// TIA Portal V17 export
// export: Created 2024-08-29T18:23:43.9089701Z, ExportSetting WithDefaults, DisplayName Totally Integrated Automation Portal, DisplayVersion V17 Update 7, DisplayName TIA Portal Openness, DisplayVersion V17 Update 7, DisplayName TIA Portal Version Control Interface, DisplayVersion V17, DisplayName SINAMICS Startdrive Advanced, DisplayVersion V17 SP2, DisplayName SINAMICS Startdrive G110M, G120, G120C, G120D, G120P, G115D, DisplayVersion V17 SP2, DisplayName SINAMICS Startdrive G130, G150, S120, S150, SINAMICS MV, S210, DisplayVersion V17 SP2, DisplayName STEP 7 Professional, DisplayVersion V17 Update 7, DisplayName STEP 7 Safety, DisplayVersion V17 Update 6, DisplayName WinCC Advanced / Unified PC, DisplayVersion V17 Update 7
FUNCTION "dcMotorControl" : Void   // FC20, LAD
{ S7_Optimized_Access := 'TRUE' }
VERSION : 0.1
// stored: AutoNumber true, IsIECCheckEnabled false, SetENOAutomatically false, UDAEnableTagReadback false
   VAR_TEMP   // added for the SCL form of the ladder/FBD networks
      _w1 : Bool;
      _w2 : Bool;
   END_VAR
BEGIN

REGION Network 1: SELECT MOTOR PARAMETERS
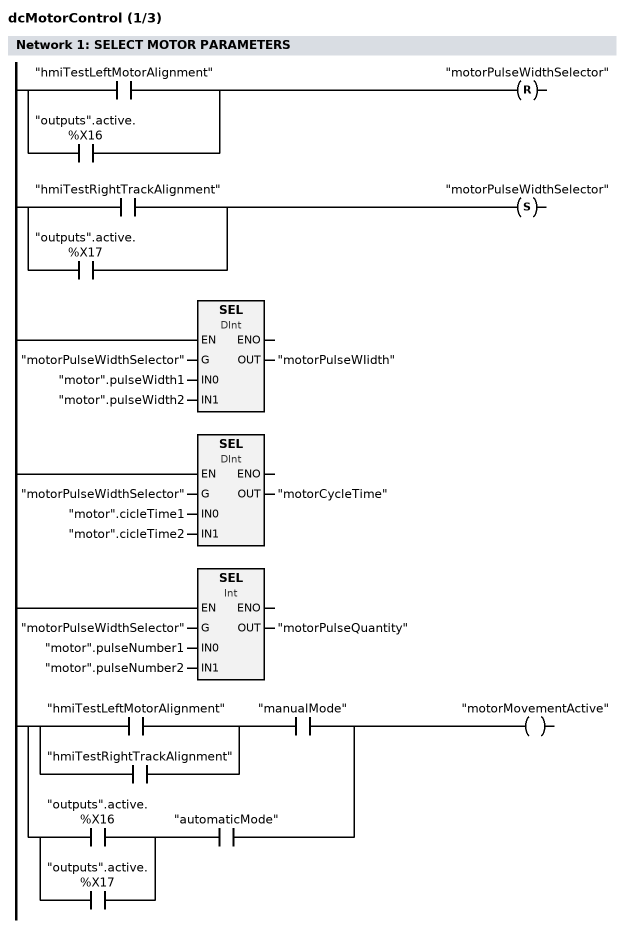
   RUNG wire#powerrail
      Contact( "hmiTestLeftMotorAlignment" )
      wire#w1
      R_Coil( "motorPulseWidthSelector" )
   END_RUNG
   RUNG wire#powerrail
      Contact( "outputs".active.%X16 )
   END_RUNG wire#w1
   RUNG wire#powerrail
      Contact( "hmiTestRightTrackAlignment" )
      wire#w2
      S_Coil( "motorPulseWidthSelector" )
   END_RUNG
   RUNG wire#powerrail
      Contact( "outputs".active.%X17 )
   END_RUNG wire#w2
   RUNG wire#powerrail
      { S7_Templates := "value_type := DInt" } SEL(g := "motorPulseWidthSelector", in0 := "motor".pulseWidth1, in1 := "motor".pulseWidth2, out => "motorPulseWIidth")
   END_RUNG
   RUNG wire#powerrail
      { S7_Templates := "value_type := DInt" } SEL(g := "motorPulseWidthSelector", in0 := "motor".cicleTime1, in1 := "motor".cicleTime2, out => "motorCycleTime")
   END_RUNG
   RUNG wire#powerrail
      { S7_Templates := "value_type := Int" } SEL(g := "motorPulseWidthSelector", in0 := "motor".pulseNumber1, in1 := "motor".pulseNumber2, out => "motorPulseQuantity")
   END_RUNG
   RUNG wire#powerrail
      Contact( "hmiTestLeftMotorAlignment" )
      wire#w3
      Contact( "manualMode" )
      wire#w4
      Coil( "motorMovementActive" )
   END_RUNG
   RUNG wire#powerrail
      Contact( "hmiTestRightTrackAlignment" )
   END_RUNG wire#w3
   RUNG wire#powerrail
      Contact( "outputs".active.%X16 )
      wire#w5
      Contact( "automaticMode" )
   END_RUNG wire#w4
   RUNG wire#powerrail
      Contact( "outputs".active.%X17 )
   END_RUNG wire#w5
   // the same network as SCL:
   IF "hmiTestLeftMotorAlignment" OR "outputs".active.%X16 THEN "motorPulseWidthSelector" := FALSE; END_IF;
   IF "hmiTestRightTrackAlignment" OR "outputs".active.%X17 THEN "motorPulseWidthSelector" := TRUE; END_IF;
   "motorPulseWIidth" := SEL(G := "motorPulseWidthSelector", IN0 := "motor".pulseWidth1, IN1 := "motor".pulseWidth2);
   "motorCycleTime" := SEL(G := "motorPulseWidthSelector", IN0 := "motor".cicleTime1, IN1 := "motor".cicleTime2);
   "motorPulseQuantity" := SEL(G := "motorPulseWidthSelector", IN0 := "motor".pulseNumber1, IN1 := "motor".pulseNumber2);
   "motorMovementActive" := (("hmiTestLeftMotorAlignment" OR "hmiTestRightTrackAlignment") AND "manualMode") OR (("outputs".active.%X16 OR "outputs".active.%X17) AND "automaticMode");
END_REGION

REGION Network 2: PWM CONTROL
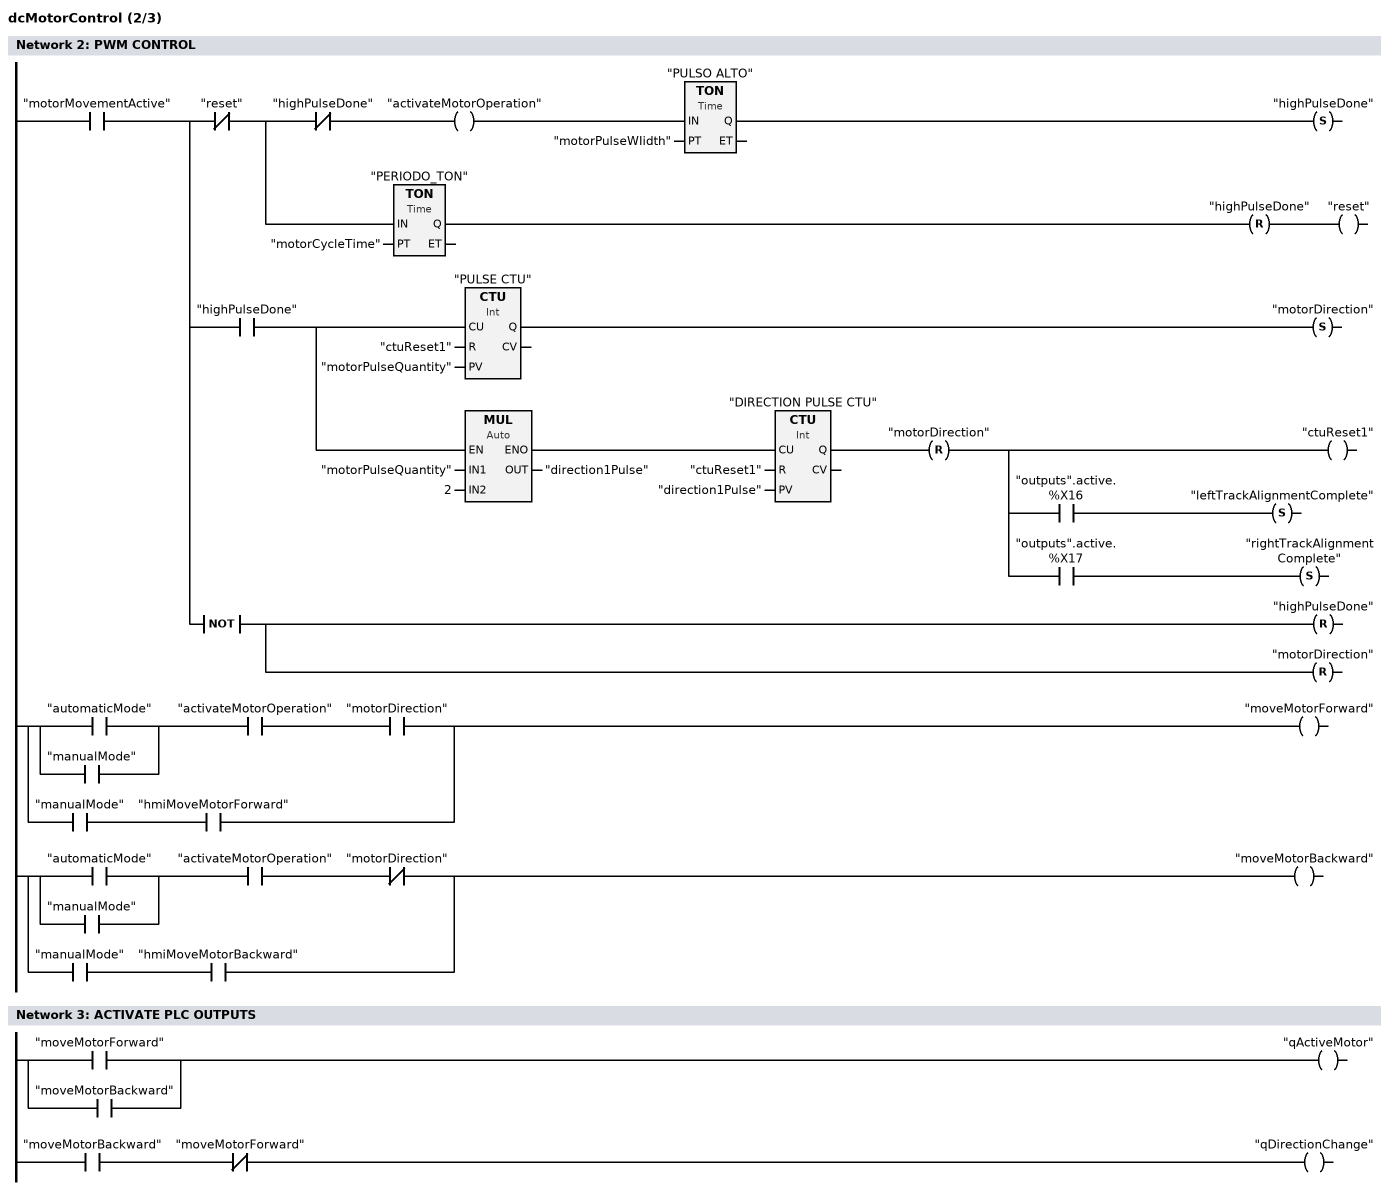
   RUNG wire#powerrail
      Contact( "motorMovementActive" )
      wire#w1
      I_Contact( "reset" )
      wire#w2
      I_Contact( "highPulseDone" )
      Coil( "activateMotorOperation" )
      { S7_Templates := "time_type := Time" } "PULSO ALTO".TON(pt := "motorPulseWIidth", et =>)
      S_Coil( "highPulseDone" )
   END_RUNG
   RUNG wire#w2
      { S7_Templates := "time_type := Time" } "PERIODO_TON".TON(pt := "motorCycleTime", et =>)
      R_Coil( "highPulseDone" )
      Coil( "reset" )
   END_RUNG
   RUNG wire#w1
      Contact( "highPulseDone" )
      wire#w3
      { S7_Templates := "value_type := Int" } "PULSE CTU".CTU(r := "ctuReset1", pv := "motorPulseQuantity", cv =>)
      S_Coil( "motorDirection" )
   END_RUNG
   RUNG wire#w3
      Mul(in1 := "motorPulseQuantity", in2 := 2, out => "direction1Pulse")
      { S7_Templates := "value_type := Int" } "DIRECTION PULSE CTU".CTU(r := "ctuReset1", pv := "direction1Pulse", cv =>)
      R_Coil( "motorDirection" )
      wire#w4
      Coil( "ctuReset1" )
   END_RUNG
   RUNG wire#w4
      Contact( "outputs".active.%X16 )
      S_Coil( "leftTrackAlignmentComplete" )
   END_RUNG
   RUNG wire#w4
      Contact( "outputs".active.%X17 )
      S_Coil( "rightTrackAlignmentComplete" )
   END_RUNG
   RUNG wire#w1
      Not()
      wire#w5
      R_Coil( "highPulseDone" )
   END_RUNG
   RUNG wire#w5
      R_Coil( "motorDirection" )
   END_RUNG
   RUNG wire#powerrail
      Contact( "automaticMode" )
      wire#w6
      Contact( "activateMotorOperation" )
      Contact( "motorDirection" )
      wire#w7
      Coil( "moveMotorForward" )
   END_RUNG
   RUNG wire#powerrail
      Contact( "manualMode" )
   END_RUNG wire#w6
   RUNG wire#powerrail
      Contact( "manualMode" )
      Contact( "hmiMoveMotorForward" )
   END_RUNG wire#w7
   RUNG wire#powerrail
      Contact( "automaticMode" )
      wire#w8
      Contact( "activateMotorOperation" )
      I_Contact( "motorDirection" )
      wire#w9
      Coil( "moveMotorBackward" )
   END_RUNG
   RUNG wire#powerrail
      Contact( "manualMode" )
   END_RUNG wire#w8
   RUNG wire#powerrail
      Contact( "manualMode" )
      Contact( "hmiMoveMotorBackward" )
   END_RUNG wire#w9
   // the same network as SCL:
   #_w1 := "motorMovementActive" AND NOT "reset";
   "activateMotorOperation" := #_w1 AND NOT "highPulseDone";
   "PULSO ALTO".TON(IN := "activateMotorOperation", PT := "motorPulseWIidth");
   IF "PULSO ALTO".Q THEN "highPulseDone" := TRUE; END_IF;
   "PERIODO_TON".TON(IN := #_w1, PT := "motorCycleTime");
   IF "PERIODO_TON".Q THEN "highPulseDone" := FALSE; END_IF;
   "reset" := "PERIODO_TON".Q;
   #_w2 := "motorMovementActive" AND "highPulseDone";
   "PULSE CTU".CTU(CU := #_w2, R := "ctuReset1", PV := "motorPulseQuantity");
   IF "PULSE CTU".Q THEN "motorDirection" := TRUE; END_IF;
   IF #_w2 THEN "direction1Pulse" := "motorPulseQuantity" * 2; END_IF;
   "DIRECTION PULSE CTU".CTU(CU := #_w2, R := "ctuReset1", PV := "direction1Pulse");
   IF "DIRECTION PULSE CTU".Q THEN "motorDirection" := FALSE; END_IF;
   "ctuReset1" := "DIRECTION PULSE CTU".Q;
   IF "DIRECTION PULSE CTU".Q AND "outputs".active.%X16 THEN "leftTrackAlignmentComplete" := TRUE; END_IF;
   IF "DIRECTION PULSE CTU".Q AND "outputs".active.%X17 THEN "rightTrackAlignmentComplete" := TRUE; END_IF;
   IF NOT "motorMovementActive" THEN
       "highPulseDone" := FALSE;
       "motorDirection" := FALSE;
   END_IF;
   "moveMotorForward" := (("automaticMode" OR "manualMode") AND "activateMotorOperation" AND "motorDirection") OR ("manualMode" AND "hmiMoveMotorForward");
   "moveMotorBackward" := (("automaticMode" OR "manualMode") AND "activateMotorOperation" AND NOT "motorDirection") OR ("manualMode" AND "hmiMoveMotorBackward");
END_REGION

REGION Network 3: ACTIVATE PLC OUTPUTS
   RUNG wire#powerrail
      Contact( "moveMotorForward" )
      wire#w1
      Coil( "qActiveMotor" )
   END_RUNG
   RUNG wire#powerrail
      Contact( "moveMotorBackward" )
   END_RUNG wire#w1
   RUNG wire#powerrail
      Contact( "moveMotorBackward" )
      I_Contact( "moveMotorForward" )
      Coil( "qDirectionChange" )
   END_RUNG
   // the same network as SCL:
   "qActiveMotor" := "moveMotorForward" OR "moveMotorBackward";
   "qDirectionChange" := "moveMotorBackward" AND NOT "moveMotorForward";
END_REGION

REGION Network 4: RESET SEQUENCER STATUS
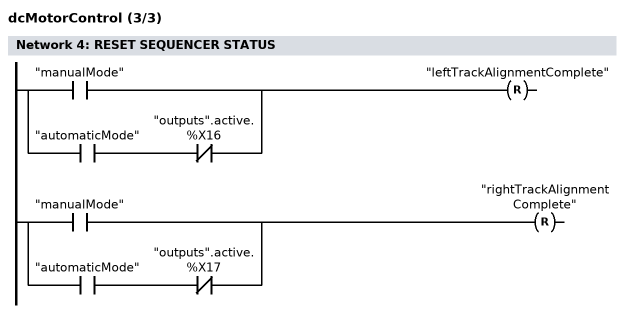
   RUNG wire#powerrail
      Contact( "manualMode" )
      wire#w1
      R_Coil( "leftTrackAlignmentComplete" )
   END_RUNG
   RUNG wire#powerrail
      Contact( "automaticMode" )
      I_Contact( "outputs".active.%X16 )
   END_RUNG wire#w1
   RUNG wire#powerrail
      Contact( "manualMode" )
      wire#w2
      R_Coil( "rightTrackAlignmentComplete" )
   END_RUNG
   RUNG wire#powerrail
      Contact( "automaticMode" )
      I_Contact( "outputs".active.%X17 )
   END_RUNG wire#w2
   // the same network as SCL:
   IF "manualMode" OR ("automaticMode" AND NOT "outputs".active.%X16) THEN
       "leftTrackAlignmentComplete" := FALSE;
   END_IF;
   IF "manualMode" OR ("automaticMode" AND NOT "outputs".active.%X17) THEN
       "rightTrackAlignmentComplete" := FALSE;
   END_IF;
END_REGION
END_FUNCTION
